// TIA Portal V20 export
TYPE "LKinCtrl_PathEditor_typePathTableExternalEvents"
// stored: Access Published
   STRUCT
      commandSelectionChanged { ExternalAccessible := 'False'; ExternalVisible := 'False'; ExternalWritable := 'False'} : Struct
         trigger : Bool;
         mode : USInt;   // 0: add, 1: edit
         command : "LKinCtrl_typePathDataElement";
      END_STRUCT;
      approachPoint { ExternalAccessible := 'False'; ExternalVisible := 'False'; ExternalWritable := 'False'} : Struct
         trigger : Bool;
         point : "LKinCtrl_typePoint";
      END_STRUCT;
      openTeachKinematics { ExternalAccessible := 'False'; ExternalVisible := 'False'; ExternalWritable := 'False'} : Bool;
      openCommandEditor { ExternalAccessible := 'False'; ExternalVisible := 'False'; ExternalWritable := 'False'} : Bool;
      closeCommandEditor { ExternalAccessible := 'False'; ExternalVisible := 'False'; ExternalWritable := 'False'} : Bool;
   END_STRUCT;
END_TYPE
